(* PLC project Pico-W v24, Unknown Unnamed 1, author Phil J *)
(* stored: creationDateTime 2024-05-07T08:00:07, contentDescription The Pico W acts as the PLC, an SH1106 OLED that use's the I2C bus (controlled by the seperate C++ script found in the "0.x: arduino_ext_0' file ) Note - unable to use the builtin led as the trigger to get the Analog value(s) This version will display both Raw and Voltage values., modificationDateTime 2024-10-09T14:30:51, language en-US *)

PROGRAM program0
  VAR
    Inp0 AT %IX0.0 : BOOL;  (* GP6 *)
    Inp1 AT %IX0.1 : BOOL;  (* GP7 *)
    Inp2 AT %IX0.2 : BOOL;  (* GP8 *)
    Inp3 AT %IX0.3 : BOOL;  (* GP9 *)
    Inp4 AT %IX0.4 : BOOL;  (* GP10 *)
    Inp5 AT %IX0.5 : BOOL;  (* GP11 *)
    Inp6 AT %IX0.6 : BOOL;  (* GP12 *)
    Inp7 AT %IX0.7 : BOOL;  (* GP13 *)
    Ana0 AT %IW0 : UINT := 0;
    Ana1 AT %IW1 : UINT := 0;
    Out1 AT %QX0.1 : BOOL;  (* GP15 *)
    Out2 AT %QX0.2 : BOOL;  (* GP16 *)
    Out3 AT %QX0.3 : BOOL;  (* GP17 *)
    Out4 AT %QX0.4 : BOOL;  (* GP18 *)
    Out5 AT %QX0.5 : BOOL;  (* GP19 *)
    Out6 AT %QX0.6 : BOOL;  (* GP20 *)
    Out7 AT %QX0.7 : BOOL;  (* GP21 *)
  END_VAR
  VAR
    Cval0 : INT := 0;
    Cval1 : INT := 0;
  END_VAR
  VAR
    Aout0 AT %QW0 : UINT := 60000;  (* GP3 Aout0 (PWM) *)
    Aout3 AT %QW3 : INT;  (* Clone of Cval0 *)
  END_VAR
  VAR
    Cout : BOOL;
    TON0 : TON;
  END_VAR
  VAR
    Out0 AT %QX0.0 : BOOL;  (* GP14 *)
  END_VAR
  VAR
    TOF0 : TOF;
    CTU0 : CTU;
    Val1 : USINT;
    Val2 : USINT;
    Val3 : USINT;
    Val4 : USINT;
    Val5 : USINT;
  END_VAR
  VAR  (* added by the conversion: wires and edge detectors of the diagram *)
    R_TRIG1 : R_TRIG;
  END_VAR

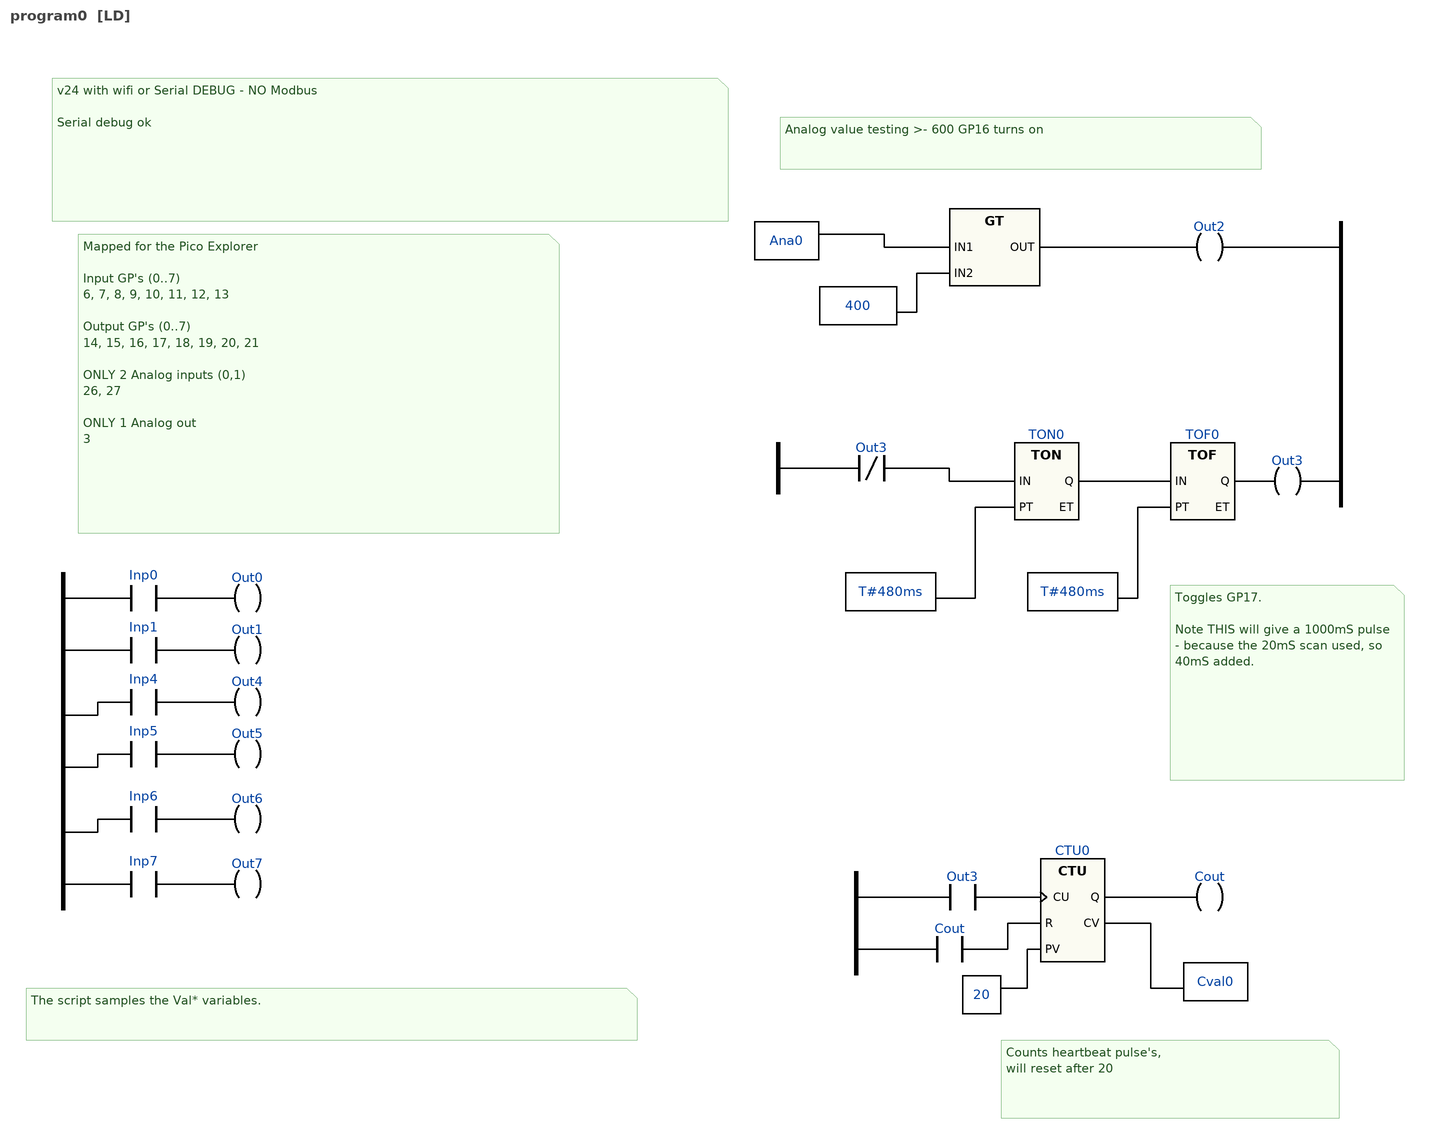
(* LD diagram, written out as Structured Text *)
(* v24 with wifi or Serial DEBUG - NO Modbus

Serial debug ok *)
(* Analog value testing >- 600 GP16 turns on *)
(* Mapped for the Pico Explorer

Input GP's (0..7)
6, 7, 8, 9, 10, 11, 12, 13

Output GP's (0..7)
14, 15, 16, 17, 18, 19, 20, 21

ONLY 2 Analog inputs (0,1)
26, 27

ONLY 1 Analog out
3 *)
Out2 := Ana0 > 400;
(* Toggles GP17.

Note THIS will give a 1000mS pulse - because the 20mS scan used, so 40mS added. *)
Out0 := Inp0;
TON0(IN := NOT Out3, PT := T#480ms);
TOF0(IN := TON0.Q, PT := T#480ms);
Out3 := TOF0.Q;
Out1 := Inp1;
Out4 := Inp4;
Out5 := Inp5;
R_TRIG1(CLK := Out3);
CTU0(CU := R_TRIG1.Q, R := Cout, PV := 20);
Cval0 := CTU0.CV;
Cout := CTU0.Q;
Out6 := Inp6;
Out7 := Inp7;
(* The script samples the Val* variables. *)
(* Counts heartbeat pulse's, 
will reset after 20 *)
END_PROGRAM

CONFIGURATION Config0
  RESOURCE Res0 ON PLC
    TASK task0(INTERVAL := T#20ms, PRIORITY := 0);
    PROGRAM instance0 WITH task0 : program0;
  END_RESOURCE
END_CONFIGURATION
